// TIA Portal project "color based pick and place seq" (V16)
// Vorlageprojekt für das Buch mit Zielsystem S7-1200

(* hardware
DEVICE "S7-1200-Station_1"  S7-1200 Station
   slot 0: "Baugruppenträger_0"  Rack  V1.0
   slot 1: "PLC_1"  CPU 1211C DC/DC/DC  6ES7 211-1AE40-0XB0  V4.1
*)

// ===== PLC "PLC_1"  CPU 1211C DC/DC/DC =====

VAR_GLOBAL   // PLC tag table "Standard-Variablentabelle"
   "start" AT %I0.0 : Bool;
   "vision" AT %IW30 : Int;
   "dif 1" AT %I0.2 : Bool;
   "box detect" AT %I0.3 : Bool;
   "z sens" AT %I0.4 : Bool;
   "x sens" AT %I0.5 : Bool;
   "emit 1" AT %Q0.0 : Bool;
   "conv1" AT %Q0.1 : Bool;
   "z down" AT %Q0.2 : Bool;
   "x move" AT %Q0.3 : Bool;
   "grab" AT %Q0.4 : Bool;
   "state" AT %MW100 : Int;
   "Tag_1" AT %M10.1 : Bool;
   "Tag_2" AT %M10.3 : Bool;
   "Tag_3" AT %M10.4 : Bool;
   "Tag_4" AT %M10.5 : Bool;
   "state dis" AT %QW30 : Int;
   "Tag_5" AT %M20.4 : Bool;
   "Tag_6" AT %M30.4 : Bool;
   "Tag_7" AT %M100.0 : Bool;
   "Tag_8" AT %M10.2 : Bool;
   "TURN LEFT" AT %Q0.5 : Bool;
   "TURN RIGHT" AT %Q0.6 : Bool;
   "TURNING" AT %I0.6 : Bool;
   "Tag_9" AT %M40.4 : Bool;
   "Tag_10" AT %M20.5 : Bool;
   "Tag_11" AT %M10.6 : Bool;
   "Tag_12" AT %M20.6 : Bool;
   "Tag_13" AT %M50.4 : Bool;
   "Tag_14" AT %M60.4 : Bool;
   "Tag_15" AT %M70.4 : Bool;
   "Tag_16" AT %M30.5 : Bool;
   "Tag_17" AT %M40.5 : Bool;
   "emit2" AT %Q0.7 : Bool;
   "emit3" AT %Q1.0 : Bool;
   "conv2" AT %Q1.1 : Bool;
   "conv3" AT %Q1.2 : Bool;
   "dif 2" AT %I0.7 : Bool;
   "diff 3" AT %I1.0 : Bool;
   "Tag_18" AT %M10.7 : Bool;
   "Tag_19" AT %M11.0 : Bool;
   "warning" AT %Q1.3 : Bool;
   "reset" AT %I0.1 : Bool;
   "last state" AT %MW102 : Int;
   "Tag_20" AT %M200.0 : Bool;
   "reset green" AT %M200.1 : Bool;
   "Tag_21" AT %M500.0 : Bool;
   "Tag_22" AT %M600.1 : Bool;
   "Tag_23" AT %M700.0 : Bool;
   "Tag_24" AT %M20.7 : Bool;
   "reset blue" AT %M200.2 : Bool;
   "Tag_25" AT %M50.5 : Bool;
   "Tag_26" AT %M30.6 : Bool;
   "Tag_27" AT %M21.0 : Bool;
END_VAR

// folder: System blocks/Program resources

DATA_BLOCK "IEC_Counter_0_DB"   // DB1
{ S7_Optimized_Access := 'TRUE' }
AUTHOR : Simatic
FAMILY : IEC
NAME : CNTR
VERSION : 1.0
// stored: InstanceOfName IEC_COUNTER
"IEC_COUNTER"
BEGIN
END_DATA_BLOCK

DATA_BLOCK "IEC_Counter_0_DB_1"   // DB2
{ S7_Optimized_Access := 'TRUE' }
AUTHOR : Simatic
FAMILY : IEC
NAME : CNTR
VERSION : 1.0
// stored: InstanceOfName IEC_COUNTER
"IEC_COUNTER"
BEGIN
END_DATA_BLOCK

DATA_BLOCK "IEC_Timer_0_DB"   // DB3
{ S7_Optimized_Access := 'TRUE' }
AUTHOR : Simatic
FAMILY : IEC
NAME : IEC_TMR
VERSION : 1.0
// stored: InstanceOfName IEC_TIMER
"IEC_TIMER"
BEGIN
END_DATA_BLOCK

DATA_BLOCK "IEC_Timer_0_DB_1"   // DB4
{ S7_Optimized_Access := 'TRUE' }
AUTHOR : Simatic
FAMILY : IEC
NAME : IEC_TMR
VERSION : 1.0
// stored: InstanceOfName IEC_TIMER
"IEC_TIMER"
BEGIN
END_DATA_BLOCK

DATA_BLOCK "IEC_Timer_0_DB_2"   // DB5
{ S7_Optimized_Access := 'TRUE' }
AUTHOR : Simatic
FAMILY : IEC
NAME : IEC_TMR
VERSION : 1.0
// stored: InstanceOfName IEC_TIMER
"IEC_TIMER"
BEGIN
END_DATA_BLOCK

DATA_BLOCK "IEC_Timer_0_DB_3"   // DB6
{ S7_Optimized_Access := 'TRUE' }
AUTHOR : Simatic
FAMILY : IEC
NAME : IEC_TMR
VERSION : 1.0
// stored: InstanceOfName IEC_TIMER
"IEC_TIMER"
BEGIN
END_DATA_BLOCK

// folder: (top level)

FUNCTION "MHJ-PLC-Lab-Function-S71200" : Void   // FC9000, SCL
{ S7_Optimized_Access := 'TRUE' }
VERSION : 0.1
   VAR_TEMP
      rdTimeReturn : Int;
      outputTime : DTL;
      SyncVal : Byte;
      forVal : Int;
      forVal_2 : Int;
      Value : Byte;
   END_VAR
   VAR CONSTANT
      CompVal : Byte := 16#34;
      Value_01 : Byte := 16#11;
      Value_01_DW : DWord := 16#A165_D992;
      Value_02_DW : DWord := 16#58BE_4401;
   END_VAR
BEGIN

   #Value:=PEEK(area := 16#82,
        dbNumber := 0,
        byteOffset := 511);
   #Value := #Value + 1;

   POKE(area := 16#82,
        dbNumber := 0,
        byteOffset := 511,
        value := #Value);

   POKE(area:=16#81,
        dbNumber:=0,
        byteOffset:=1016,
        value:=#Value_01_DW);
   POKE(area := 16#81,
        dbNumber := 0,
        byteOffset := 1020,
        value := #Value_02_DW);

   POKE(area := 16#81,
        dbNumber := 0,
        byteOffset := 511,
        value := B#16#00);

   FOR #forVal := 0 TO 120 DO
       FOR #forVal_2:=0 TO 10 DO
           #rdTimeReturn:=RD_SYS_T(#outputTime);
           #rdTimeReturn := WR_SYS_T(#outputTime);
           #rdTimeReturn := RD_SYS_T(#outputTime);
           #rdTimeReturn := WR_SYS_T(#outputTime);
       END_FOR;
       #SyncVal:= PEEK(area := 16#81,
                      dbNumber := 0,
                      byteOffset := 511);
       IF #SyncVal = #CompVal THEN
          GOTO M_1;
       END_IF;
   END_FOR;
   RETURN;

   M_1:
   POKE(area := 16#81,
        dbNumber := 0,
        byteOffset := 511,
        value := B#16#0);
END_FUNCTION

ORGANIZATION_BLOCK "Main"   // OB1, LAD, ProgramCycle
TITLE = "Main Program Sweep (Cycle)"
{ S7_Optimized_Access := 'TRUE' }
VERSION : 0.1
   VAR_INPUT
      Initial_Call : Bool;   // Initial call of this OB
      Remanence : Bool;   // =True, if remanent data are available
   END_VAR
   VAR_TEMP   // added for the SCL form of the ladder/FBD networks
      _w1 : Bool;
      _w2 : Bool;
      _w3 : Bool;
      _w4 : Bool;
      _w5 : Bool;
      _w6 : Bool;
      _w7 : Bool;
      _w8 : Bool;
      _w9 : Bool;
   END_VAR
BEGIN

REGION Network 1
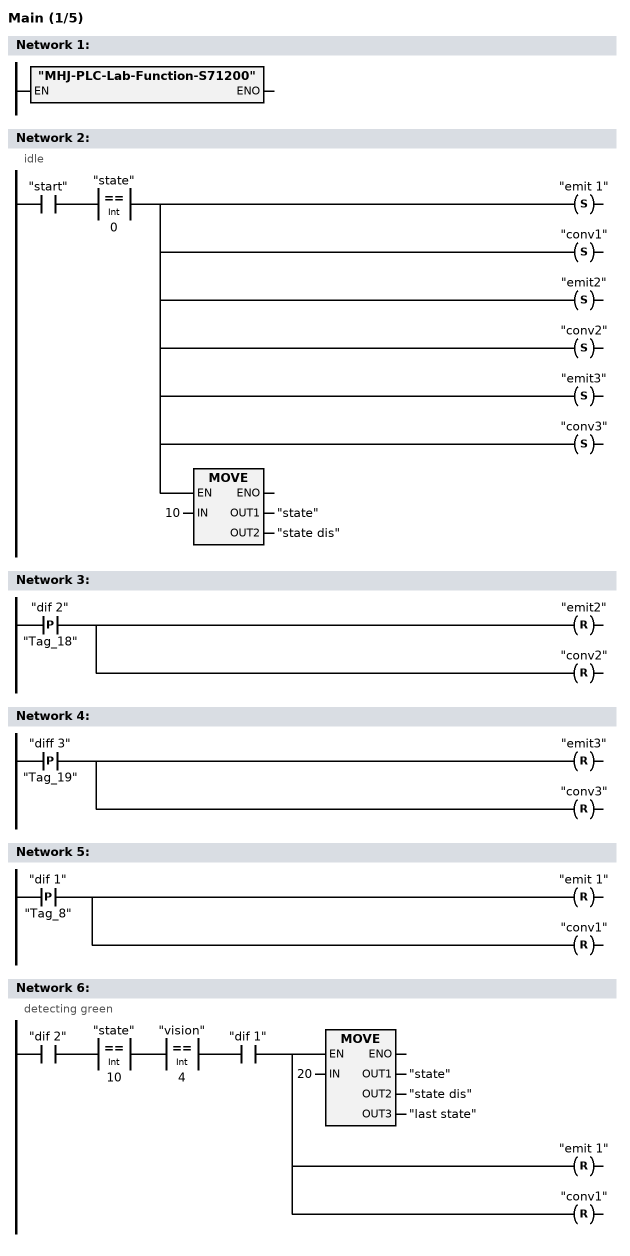
   RUNG wire#powerrail
      "MHJ-PLC-Lab-Function-S71200"()
   END_RUNG
   // the same network as SCL:
   "MHJ-PLC-Lab-Function-S71200"();
END_REGION

REGION Network 2
   // idle
   RUNG wire#powerrail
      Contact( "start" )
      { S7_Templates := "SrcType := Int" } EQ_Contact(in1 := "state", in2 := 0)
      wire#w1
      S_Coil( "emit 1" )
   END_RUNG
   RUNG wire#w1
      S_Coil( "conv1" )
   END_RUNG
   RUNG wire#w1
      S_Coil( "emit2" )
   END_RUNG
   RUNG wire#w1
      S_Coil( "conv2" )
   END_RUNG
   RUNG wire#w1
      S_Coil( "emit3" )
   END_RUNG
   RUNG wire#w1
      S_Coil( "conv3" )
   END_RUNG
   RUNG wire#w1
      Move(in := 10, out1 => "state", out2 => "state dis")
   END_RUNG
   // the same network as SCL:
   IF "start" AND ("state" = 0) THEN
       "emit 1" := TRUE;
       "conv1" := TRUE;
       "emit2" := TRUE;
       "conv2" := TRUE;
       "emit3" := TRUE;
       "conv3" := TRUE;
       "state" := 10;
       "state dis" := 10;
   END_IF;
END_REGION

REGION Network 3
   RUNG wire#powerrail
      P_Contact(operand := "dif 2", bit := "Tag_18")
      wire#w1
      R_Coil( "emit2" )
   END_RUNG
   RUNG wire#w1
      R_Coil( "conv2" )
   END_RUNG
   // the same network as SCL:
   #_w1 := "dif 2" AND NOT "Tag_18";   // rising edge of "dif 2"
   "Tag_18" := "dif 2";
   IF #_w1 THEN
       "emit2" := FALSE;
       "conv2" := FALSE;
   END_IF;
END_REGION

REGION Network 4
   RUNG wire#powerrail
      P_Contact(operand := "diff 3", bit := "Tag_19")
      wire#w1
      R_Coil( "emit3" )
   END_RUNG
   RUNG wire#w1
      R_Coil( "conv3" )
   END_RUNG
   // the same network as SCL:
   #_w1 := "diff 3" AND NOT "Tag_19";   // rising edge of "diff 3"
   "Tag_19" := "diff 3";
   IF #_w1 THEN
       "emit3" := FALSE;
       "conv3" := FALSE;
   END_IF;
END_REGION

REGION Network 5
   RUNG wire#powerrail
      P_Contact(operand := "dif 1", bit := "Tag_8")
      wire#w1
      R_Coil( "emit 1" )
   END_RUNG
   RUNG wire#w1
      R_Coil( "conv1" )
   END_RUNG
   // the same network as SCL:
   #_w1 := "dif 1" AND NOT "Tag_8";   // rising edge of "dif 1"
   "Tag_8" := "dif 1";
   IF #_w1 THEN
       "emit 1" := FALSE;
       "conv1" := FALSE;
   END_IF;
END_REGION

REGION Network 6
   // detecting green
   RUNG wire#powerrail
      Contact( "dif 2" )
      { S7_Templates := "SrcType := Int" } EQ_Contact(in1 := "state", in2 := 10)
      { S7_Templates := "SrcType := Int" } EQ_Contact(in1 := "vision", in2 := 4)
      Contact( "dif 1" )
      wire#w1
      Move(in := 20, out1 => "state", out2 => "state dis", out3 => "last state")
   END_RUNG
   RUNG wire#w1
      R_Coil( "emit 1" )
   END_RUNG
   RUNG wire#w1
      R_Coil( "conv1" )
   END_RUNG
   // the same network as SCL:
   #_w1 := "dif 2" AND ("state" = 10) AND ("vision" = 4) AND "dif 1";
   IF #_w1 THEN
       "state" := 20;
       "state dis" := 20;
       "last state" := 20;
       "emit 1" := FALSE;
       "conv1" := FALSE;
   END_IF;
END_REGION

REGION Network 7
   // detecting blue
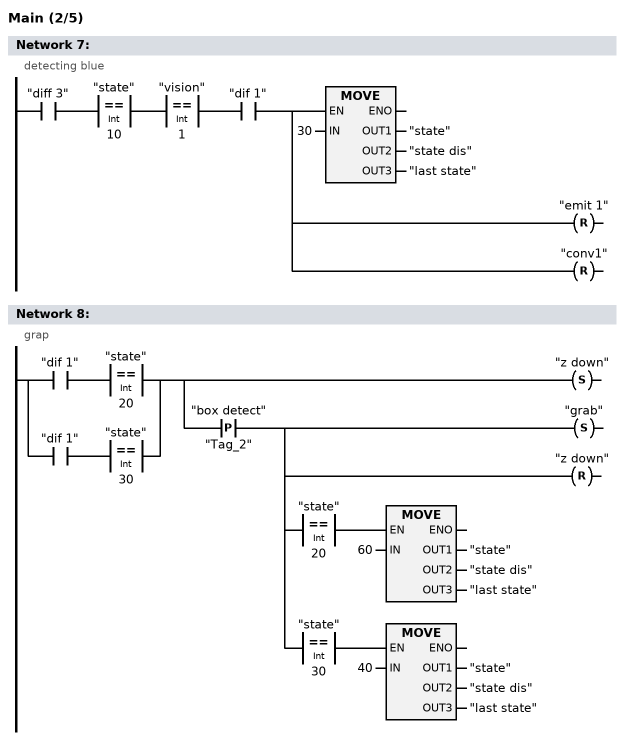
   RUNG wire#powerrail
      Contact( "diff 3" )
      { S7_Templates := "SrcType := Int" } EQ_Contact(in1 := "state", in2 := 10)
      { S7_Templates := "SrcType := Int" } EQ_Contact(in1 := "vision", in2 := 1)
      Contact( "dif 1" )
      wire#w1
      Move(in := 30, out1 => "state", out2 => "state dis", out3 => "last state")
   END_RUNG
   RUNG wire#w1
      R_Coil( "emit 1" )
   END_RUNG
   RUNG wire#w1
      R_Coil( "conv1" )
   END_RUNG
   // the same network as SCL:
   #_w1 := "diff 3" AND ("state" = 10) AND ("vision" = 1) AND "dif 1";
   IF #_w1 THEN
       "state" := 30;
       "state dis" := 30;
       "last state" := 30;
       "emit 1" := FALSE;
       "conv1" := FALSE;
   END_IF;
END_REGION

REGION Network 8
   // grap
   RUNG wire#powerrail
      Contact( "dif 1" )
      { S7_Templates := "SrcType := Int" } EQ_Contact(in1 := "state", in2 := 20)
      wire#w1
      S_Coil( "z down" )
   END_RUNG
   RUNG wire#powerrail
      Contact( "dif 1" )
      { S7_Templates := "SrcType := Int" } EQ_Contact(in1 := "state", in2 := 30)
   END_RUNG wire#w1
   RUNG wire#w1
      P_Contact(operand := "box detect", bit := "Tag_2")
      wire#w2
      S_Coil( "grab" )
   END_RUNG
   RUNG wire#w2
      R_Coil( "z down" )
   END_RUNG
   RUNG wire#w2
      { S7_Templates := "SrcType := Int" } EQ_Contact(in1 := "state", in2 := 20)
      Move(in := 60, out1 => "state", out2 => "state dis", out3 => "last state")
   END_RUNG
   RUNG wire#w2
      { S7_Templates := "SrcType := Int" } EQ_Contact(in1 := "state", in2 := 30)
      Move(in := 40, out1 => "state", out2 => "state dis", out3 => "last state")
   END_RUNG
   // the same network as SCL:
   #_w1 := ("dif 1" AND ("state" = 20)) OR ("dif 1" AND ("state" = 30));
   IF #_w1 THEN "z down" := TRUE; END_IF;
   #_w2 := #_w1 AND "box detect" AND NOT "Tag_2";   // rising edge of "box detect"
   "Tag_2" := "box detect";
   IF #_w2 THEN
       "grab" := TRUE;
       "z down" := FALSE;
   END_IF;
   IF #_w2 AND ("state" = 20) THEN
       "state" := 60;
       "state dis" := 60;
       "last state" := 60;
   END_IF;
   IF #_w2 AND ("state" = 30) THEN
       "state" := 40;
       "state dis" := 40;
       "last state" := 40;
   END_IF;
END_REGION

REGION Network 9
   // green
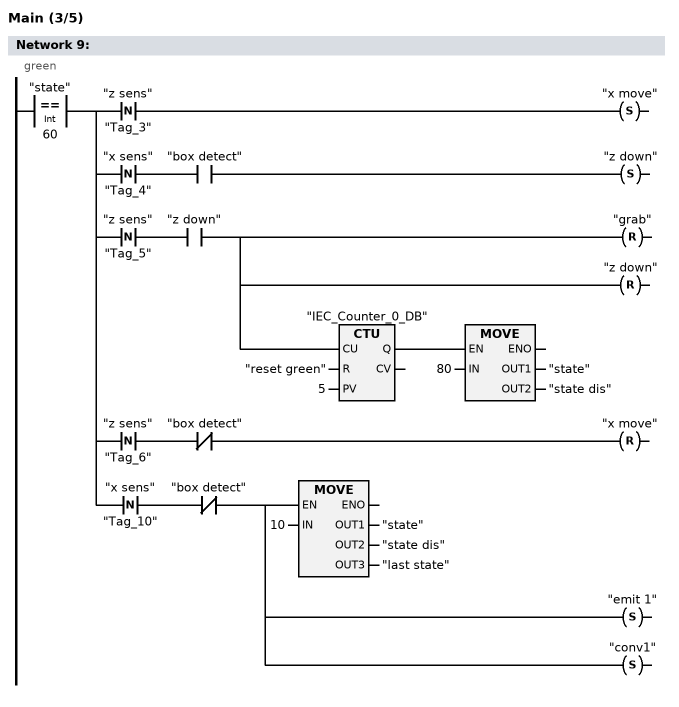
   #_w1 := "state" = 60;
   #_w2 := #_w1 AND NOT "z sens" AND "Tag_3";   // falling edge of "z sens"
   "Tag_3" := "z sens";
   IF #_w2 THEN "x move" := TRUE; END_IF;
   #_w3 := #_w1 AND NOT "x sens" AND "Tag_4";   // falling edge of "x sens"
   "Tag_4" := "x sens";
   IF #_w3 AND "box detect" THEN "z down" := TRUE; END_IF;
   #_w4 := #_w1 AND NOT "z sens" AND "Tag_5";   // falling edge of "z sens"
   "Tag_5" := "z sens";
   #_w5 := #_w4 AND "z down";
   IF #_w5 THEN
       "grab" := FALSE;
       "z down" := FALSE;
   END_IF;
   "IEC_Counter_0_DB".CTU(CU := #_w5, R := "reset green", PV := 5);
   IF "IEC_Counter_0_DB".Q THEN
       "state" := 80;
       "state dis" := 80;
   END_IF;
   #_w6 := #_w1 AND NOT "z sens" AND "Tag_6";   // falling edge of "z sens"
   "Tag_6" := "z sens";
   IF #_w6 AND NOT "box detect" THEN "x move" := FALSE; END_IF;
   #_w7 := #_w1 AND NOT "x sens" AND "Tag_10";   // falling edge of "x sens"
   "Tag_10" := "x sens";
   IF #_w7 AND NOT "box detect" THEN
       "state" := 10;
       "state dis" := 10;
       "last state" := 10;
       "emit 1" := TRUE;
       "conv1" := TRUE;
   END_IF;
END_REGION

REGION Network 10
   // blue
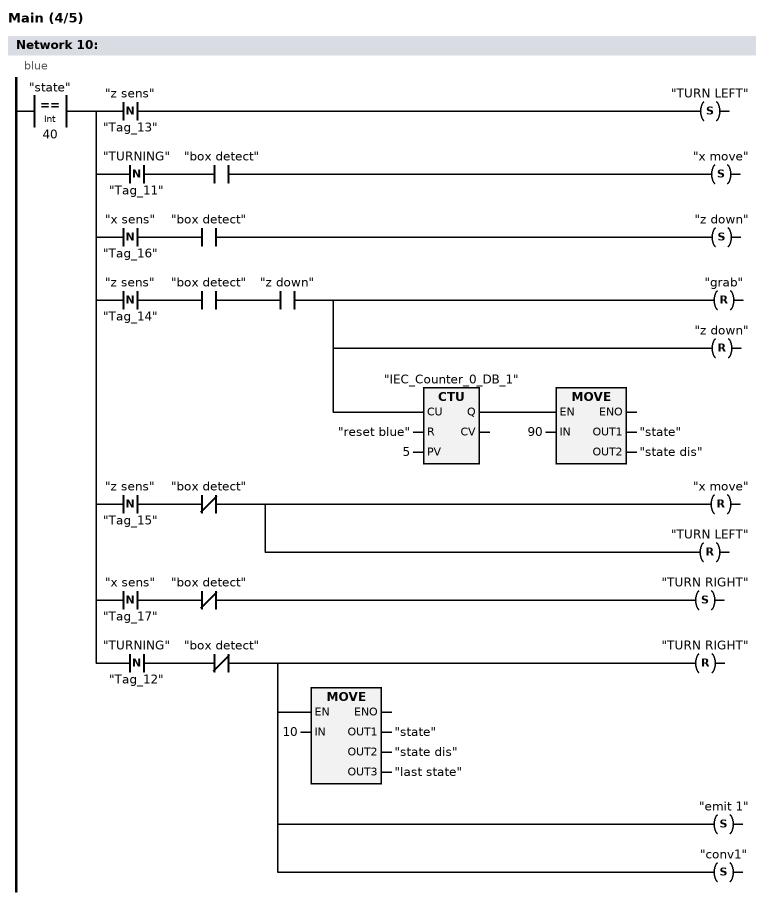
   #_w1 := "state" = 40;
   #_w2 := #_w1 AND NOT "z sens" AND "Tag_13";   // falling edge of "z sens"
   "Tag_13" := "z sens";
   IF #_w2 THEN "TURN LEFT" := TRUE; END_IF;
   #_w3 := #_w1 AND NOT "TURNING" AND "Tag_11";   // falling edge of "TURNING"
   "Tag_11" := "TURNING";
   IF #_w3 AND "box detect" THEN "x move" := TRUE; END_IF;
   #_w4 := #_w1 AND NOT "x sens" AND "Tag_16";   // falling edge of "x sens"
   "Tag_16" := "x sens";
   IF #_w4 AND "box detect" THEN "z down" := TRUE; END_IF;
   #_w5 := #_w1 AND NOT "z sens" AND "Tag_14";   // falling edge of "z sens"
   "Tag_14" := "z sens";
   #_w6 := #_w5 AND "box detect" AND "z down";
   IF #_w6 THEN
       "grab" := FALSE;
       "z down" := FALSE;
   END_IF;
   "IEC_Counter_0_DB_1".CTU(CU := #_w6, R := "reset blue", PV := 5);
   IF "IEC_Counter_0_DB_1".Q THEN
       "state" := 90;
       "state dis" := 90;
   END_IF;
   #_w7 := #_w1 AND NOT "z sens" AND "Tag_15";   // falling edge of "z sens"
   "Tag_15" := "z sens";
   IF #_w7 AND NOT "box detect" THEN
       "x move" := FALSE;
       "TURN LEFT" := FALSE;
   END_IF;
   #_w8 := #_w1 AND NOT "x sens" AND "Tag_17";   // falling edge of "x sens"
   "Tag_17" := "x sens";
   IF #_w8 AND NOT "box detect" THEN "TURN RIGHT" := TRUE; END_IF;
   #_w9 := #_w1 AND NOT "TURNING" AND "Tag_12";   // falling edge of "TURNING"
   "Tag_12" := "TURNING";
   IF #_w9 AND NOT "box detect" THEN
       "TURN RIGHT" := FALSE;
       "state" := 10;
       "state dis" := 10;
       "last state" := 10;
       "emit 1" := TRUE;
       "conv1" := TRUE;
   END_IF;
END_REGION

REGION Network 11
   // reset
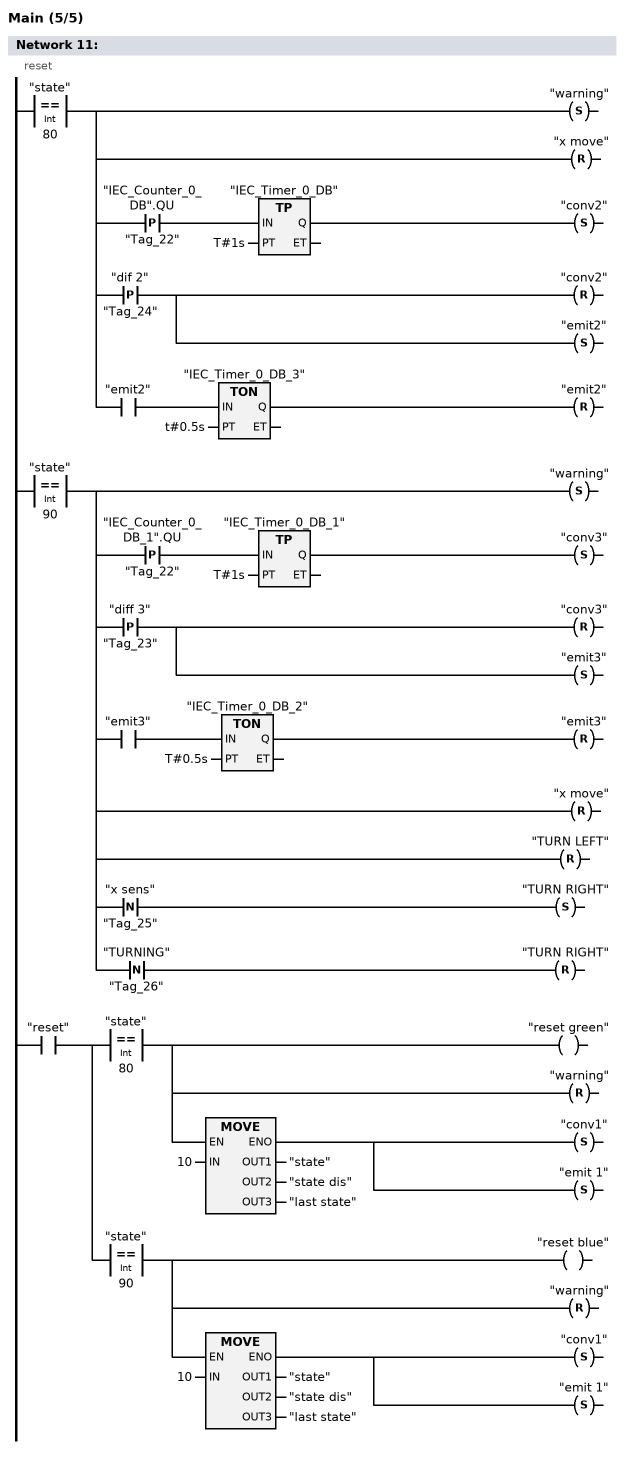
   #_w1 := "state" = 80;
   IF #_w1 THEN
       "warning" := TRUE;
       "x move" := FALSE;
   END_IF;
   #_w2 := #_w1 AND "IEC_Counter_0_DB".QU AND NOT "Tag_22";   // rising edge of "IEC_Counter_0_DB".QU
   "Tag_22" := "IEC_Counter_0_DB".QU;
   "IEC_Timer_0_DB".TP(IN := #_w2, PT := T#1s);
   IF "IEC_Timer_0_DB".Q THEN "conv2" := TRUE; END_IF;
   #_w3 := #_w1 AND "dif 2" AND NOT "Tag_24";   // rising edge of "dif 2"
   "Tag_24" := "dif 2";
   IF #_w3 THEN
       "conv2" := FALSE;
       "emit2" := TRUE;
   END_IF;
   "IEC_Timer_0_DB_3".TON(IN := #_w1 AND "emit2", PT := t#0.5s);
   IF "IEC_Timer_0_DB_3".Q THEN "emit2" := FALSE; END_IF;
   #_w4 := "state" = 90;
   IF #_w4 THEN "warning" := TRUE; END_IF;
   #_w5 := #_w4 AND "IEC_Counter_0_DB_1".QU AND NOT "Tag_22";   // rising edge of "IEC_Counter_0_DB_1".QU
   "Tag_22" := "IEC_Counter_0_DB_1".QU;
   "IEC_Timer_0_DB_1".TP(IN := #_w5, PT := T#1s);
   IF "IEC_Timer_0_DB_1".Q THEN "conv3" := TRUE; END_IF;
   #_w6 := #_w4 AND "diff 3" AND NOT "Tag_23";   // rising edge of "diff 3"
   "Tag_23" := "diff 3";
   IF #_w6 THEN
       "conv3" := FALSE;
       "emit3" := TRUE;
   END_IF;
   "IEC_Timer_0_DB_2".TON(IN := #_w4 AND "emit3", PT := T#0.5s);
   IF "IEC_Timer_0_DB_2".Q THEN "emit3" := FALSE; END_IF;
   IF #_w4 THEN
       "x move" := FALSE;
       "TURN LEFT" := FALSE;
   END_IF;
   #_w7 := #_w4 AND NOT "x sens" AND "Tag_25";   // falling edge of "x sens"
   "Tag_25" := "x sens";
   IF #_w7 THEN "TURN RIGHT" := TRUE; END_IF;
   #_w8 := #_w4 AND NOT "TURNING" AND "Tag_26";   // falling edge of "TURNING"
   "Tag_26" := "TURNING";
   IF #_w8 THEN "TURN RIGHT" := FALSE; END_IF;
   "reset green" := "reset" AND ("state" = 80);
   IF "reset green" THEN
       "warning" := FALSE;
       "state" := 10;
       "state dis" := 10;
       "last state" := 10;
       "conv1" := TRUE;
       "emit 1" := TRUE;
   END_IF;
   "reset blue" := "reset" AND ("state" = 90);
   IF "reset blue" THEN
       "warning" := FALSE;
       "state" := 10;
       "state dis" := 10;
       "last state" := 10;
       "conv1" := TRUE;
       "emit 1" := TRUE;
   END_IF;
END_REGION
END_ORGANIZATION_BLOCK